FUNCTION_BLOCK SingleASingleE (* Template for an empty basic function block *)
  (* Standard: 61499-2; Description: Copyright (c) 2019 Jan Holzweber This program and the accompanying materials are made available under the terms of the Eclipse Public License 2.0 which is available at https://www.eclipse.org/legal/epl-2.0/ SPDX-License-Identifier: EPL-2.0 *)
  (* Version 1.0, 2019-06-11, Jan Holzweber *)
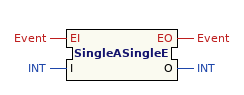
  EVENT_INPUT
    EI;
  END_EVENT
  EVENT_OUTPUT
    EO;
  END_EVENT
  VAR_INPUT
    I : INT;
  END_VAR
  VAR_OUTPUT
    O : INT;
  END_VAR
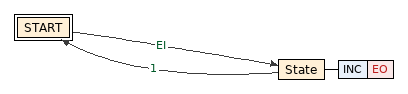
  EC_STATES
    START; (* Initial State *)
    State : INC -> EO;
  END_STATES
  EC_TRANSITIONS
    START TO State := EI;
    State TO START := 1;
  END_TRANSITIONS
  ALGORITHM INC IN ST: (* new algorithm *)
O:=I+1;
  END_ALGORITHM
END_FUNCTION_BLOCK
